TEXTLIST EL1809_S_1
  1 = 'Altimetric limit' | chinese: '探块限位' | Chinese: '探块限位'
  2 = 'Z Axis origin' | chinese: 'Z轴原点' | Chinese: 'Z轴原点'
  3 = 'Z Axis limitP' | chinese: 'Z轴下极限' | Chinese: 'Z轴下极限'
  4 = 'SubInkTankLevel C1' | chinese: '二级墨盒液位C1' | Chinese: '二级墨盒液位C1'
  5 = 'SubInkTankLevel C2' | chinese: '二级墨盒液位C2' | Chinese: '二级墨盒液位C2'
  6 = 'SubInkTankLevel Y1' | chinese: '二级墨盒液位Y1' | Chinese: '二级墨盒液位Y1'
  7 = 'SubInkTankLevel Y2' | chinese: '二级墨盒液位Y2' | Chinese: '二级墨盒液位Y2'
  8 = 'SubInkTankLevel M1' | chinese: '二级墨盒液位M1' | Chinese: '二级墨盒液位M1'
  9 = 'SubInkTankLevel M2' | chinese: '二级墨盒液位M2' | Chinese: '二级墨盒液位M2'
  10 = 'SubInkTankLevel K1' | chinese: '二级墨盒液位K1' | Chinese: '二级墨盒液位K1'
  11 = 'SubInkTankLevel K2' | chinese: '二级墨盒液位K2' | Chinese: '二级墨盒液位K2'
  12 = 'SubInkTankLevel LC1' | chinese: '二级墨盒液位LC1' | Chinese: '二级墨盒液位LC1'
  13 = 'SubInkTankLevel LC2' | chinese: '二级墨盒液位LC2' | Chinese: '二级墨盒液位LC2'
  14 = 'SubInkTankLevel LM1' | chinese: '二级墨盒液位LM1' | Chinese: '二级墨盒液位LM1'
  15 = 'SubInkTankLevel LM2' | chinese: '二级墨盒液位LM2' | Chinese: '二级墨盒液位LM2'
  16 = 'SubInkTankLevel P1' | chinese: '二级墨盒液位图层1' | Chinese: '二级墨盒液位图层1'
   = ''
END_TEXTLIST

(* stored: Version 1.1.0.1, ProductVersion 3.1.4024.11
   TextList EL1809_S_1: Id {6347fd89-2cf3-43b6-8b97-c420ab72f580} *)
